Fanuc KAREL source: kb00027.KL

-- PROVISIONAL review KL for V770-1; original PC SHA256 3bdf697414d766ec9ad19ce69c44b7395fcdf9e426d07ba49306700fb56d97c6
-- Incomplete behavior may be omitted. Consult companion uncertainty JSON. Do not deploy.
PROGRAM KB00027
%NOLOCKGROUP
BEGIN
  -- UNRESOLVED_PC offsets 5-12; opcodes 9D,23
  -- UNRESOLVED_PC offsets 17-26; opcodes 3F,75
  -- UNRESOLVED_PC offsets 31-38; opcodes 9D,23
  -- UNRESOLVED_PC offsets 43-67; opcodes 27,22,22,2A,22,31
  -- UNRESOLVED_PC offsets 72-76; opcodes 7F
END KB00027
